% RSLogix 500 project SW2046_W.RSS, saved by version 11.00.00.00 %
PROJECT "PS7"    % processor: MicroLogix 1400 %

PROGRAM FILES
  LAD 2 "MAIN"  33 rungs  % Calls all system and subsystem routines %
  LAD 3 "CONSTANTS"  90 rungs  % Maintains the system constants %
  LAD 4 "DEFAULTS"  121 rungs  % Manages the system default values %
  LAD 5 "SYS_FAULTS"  58 rungs  % Monitors the system fault conditions %
  LAD 6 "SYSTEM"  93 rungs  % Controls the system %
  LAD 7 "PROCESSING"  14 rungs  % Runs the processing control %
  LAD 8 "MANUAL_CTL"  17 rungs  % Runs the manual valve control %
  LAD 9 "STARTUP"  25 rungs
  LAD 10 "PURIFY"  38 rungs  % Operates the purify control %
  LAD 11 "REGEN"  55 rungs  % Operates the regen control %
  LAD 12 "REGEN_FLT"  26 rungs  % regen alarms and warnings %
  LAD 13 "PURGE"  34 rungs
  LAD 14 "MFM"  5 rungs
  LAD 16 "MFC"  12 rungs
  LAD 17 "BYPASS"  4 rungs  % Controls the bypass %
  LAD 20 "ADS A"  46 rungs  % Controls the Adsorber A %
  LAD 21 "ADS A FLT"  18 rungs  % Controls the Adsorber A faults %
  LAD 22 "ADS B"  46 rungs  % Controld Adsorber B %
  LAD 23 "ADS B FLT"  17 rungs  % Controls the Adsorber B faults %
  LAD 24 "ADS PH"  10 rungs
  LAD 25 "ADS PH FLT"  15 rungs
  LAD 26 "GETTER"  24 rungs
  LAD 27 "GET 1 FLT"  15 rungs
  LAD 28 "GET 1"  25 rungs
  LAD 29 "GET 2 FLT"  15 rungs
  LAD 30 "GET 2"  25 rungs
  LAD 31 "GET 3 FLT"  15 rungs
  LAD 32 "GET 3"  25 rungs
  LAD 49 "MODBUS"  59 rungs
  LAD 50 "PLC FAULT"  7 rungs
  LAD 51 "REVERSE"  9 rungs
  LAD 252 "CLR_0034"  8 rungs

DATA FILES
  O0 OUTPUT  40 elements
  I1 INPUT  41 elements
  S2 STATUS  66 elements
  B3 BINARY  4 elements
  T4 TIMER  256 elements
  C5 COUNTER  256 elements
  R6 CONTROL  2 elements
  N7 SYSTEM CFG  120 elements  % Maintains the values that characterize the system %
  F8 FLOAT  8 elements
  N9 CONSTANTS  124 elements  % The collection of system and subsystem constants %
  N10 SYSTEM  36 elements  % Contain the values for system control %
  N11 PROCESS  4 elements  % Contains the values for the processing machine %
  N12 PURIFY  18 elements  % Contains the values required for purify %
  N13 REGEN  32 elements  % Contains the values required for regen %
  PD14 PID  10 elements
  N15 MANUAL CTL  5 elements  % Contains the data for the manual valve control %
  N16 ADSORBER_A  22 elements  % Contains the values for Adsorber A %
  N17 ADSORBER_B  22 elements  % Contains the values required for Adsorber B %
  N18 GETTER CMN  28 elements
  N19 BYPASS  2 elements
  N20 PURGE  10 elements
  N21 STARTUP  80 elements
  B22 STARTUP  6 elements
  N23 GETTER 1  15 elements
  N24 GETTER 2  15 elements
  N25 GETTER 3  15 elements
  B26 FAULTS  29 elements
  N27 NOMEMBCKUP  3 elements
  B29 GETTER  1 elements
  B30 SYSTEM CFG  6 elements
  B31 SYSTEM  10 elements
  B32 PROCESS  1 elements
  B33 PURIFY  1 elements
  B34 REGEN  3 elements
  B35 MANUAL CTL  3 elements
  B36 PURGE  2 elements
  L51 LONG  4 elements
  N55 TEST_START  5 elements  % Simultation Start %
  N64 MODBUS  126 elements
  MG68 COMMS  2 elements
  B69 REVERSE  3 elements
  N77 FAULT_FIFO  255 elements
  RIX81   1 elements
  N200   1 elements
  L201   1 elements
  L202   1 elements
  L203   2 elements
  F206   3 elements
  N207   6 elements
  N210   3 elements
  B250   1 elements
  T252   5 elements
  C253   6 elements

LADDER 2 "MAIN"    % Calls all system and subsystem routines %
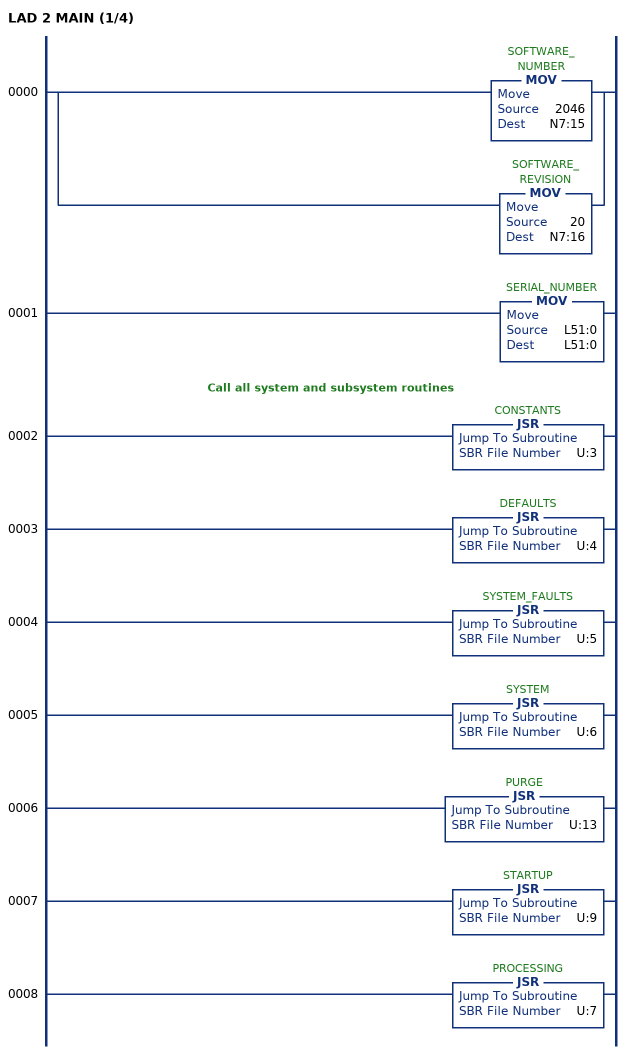
% Rung: 0 %
SOR BST MOV 2046 N7:15 NXB MOV 20 N7:16 BND EOR
%   N7:15  SOFTWARE_NUMBER %
%   N7:16  SOFTWARE_REVISION %
% Rung: 1 %
SOR MOV L51:0 L51:0 EOR
%   L51:0  SERIAL_NUMBER %
% Rung: 2 %
% TITLE: Call all system and subsystem routines %
SOR JSR U:3 EOR
%   U:3  CONSTANTS %
% Rung: 3 %
SOR JSR U:4 EOR
%   U:4  DEFAULTS %
% Rung: 4 %
SOR JSR U:5 EOR
%   U:5  SYSTEM_FAULTS %
% Rung: 5 %
SOR JSR U:6 EOR
%   U:6  SYSTEM %
% Rung: 6 %
SOR JSR U:13 EOR
%   U:13  PURGE %
% Rung: 7 %
SOR JSR U:9 EOR
%   U:9  STARTUP %
% Rung: 8 %
SOR JSR U:7 EOR
%   U:7  PROCESSING %

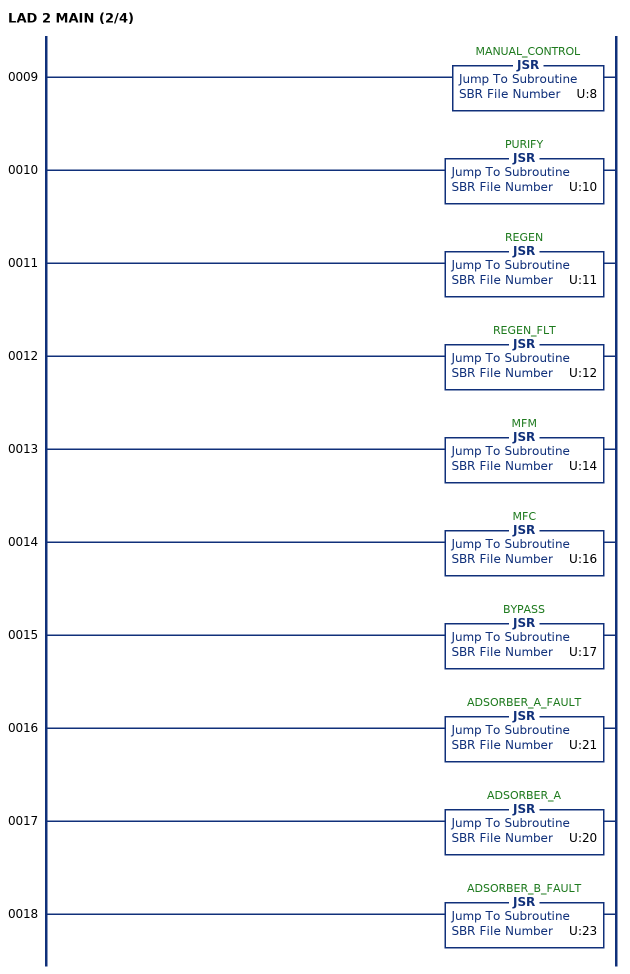
% Rung: 9 %
SOR JSR U:8 EOR
%   U:8  MANUAL_CONTROL %
% Rung: 10 %
SOR JSR U:10 EOR
%   U:10  PURIFY %
% Rung: 11 %
SOR JSR U:11 EOR
%   U:11  REGEN %
% Rung: 12 %
SOR JSR U:12 EOR
%   U:12  REGEN_FLT %
% Rung: 13 %
SOR JSR U:14 EOR
%   U:14  MFM %
% Rung: 14 %
SOR JSR U:16 EOR
%   U:16  MFC %
% Rung: 15 %
SOR JSR U:17 EOR
%   U:17  BYPASS %
% Rung: 16 %
SOR JSR U:21 EOR
%   U:21  ADSORBER_A_FAULT %
% Rung: 17 %
SOR JSR U:20 EOR
%   U:20  ADSORBER_A %
% Rung: 18 %
SOR JSR U:23 EOR
%   U:23  ADSORBER_B_FAULT %

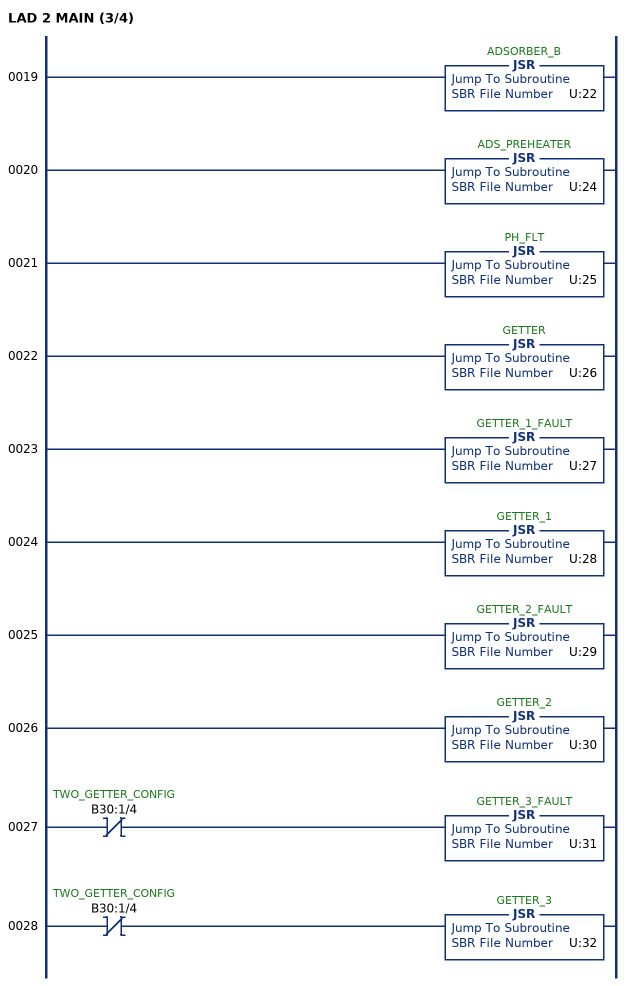
% Rung: 19 %
SOR JSR U:22 EOR
%   U:22  ADSORBER_B %
% Rung: 20 %
SOR JSR U:24 EOR
%   U:24  ADS_PREHEATER %
% Rung: 21 %
SOR JSR U:25 EOR
%   U:25  PH_FLT %
% Rung: 22 %
SOR JSR U:26 EOR
%   U:26  GETTER %
% Rung: 23 %
SOR JSR U:27 EOR
%   U:27  GETTER_1_FAULT %
% Rung: 24 %
SOR JSR U:28 EOR
%   U:28  GETTER_1 %
% Rung: 25 %
SOR JSR U:29 EOR
%   U:29  GETTER_2_FAULT %
% Rung: 26 %
SOR JSR U:30 EOR
%   U:30  GETTER_2 %
% Rung: 27 %
SOR XIO B30:1/4 JSR U:31 EOR
%   B30:1/4  TWO_GETTER_CONFIG %
%   U:31  GETTER_3_FAULT %
% Rung: 28 %
SOR XIO B30:1/4 JSR U:32 EOR
%   B30:1/4  TWO_GETTER_CONFIG %
%   U:32  GETTER_3 %

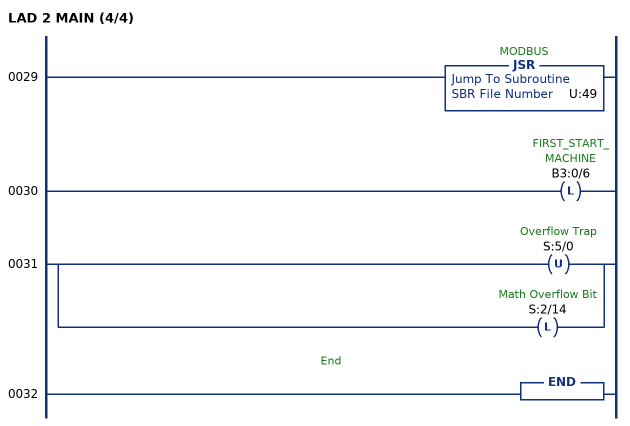
% Rung: 29 %
SOR JSR U:49 EOR
%   U:49  MODBUS %
% Rung: 30 %
SOR OTL B3:0/6 EOR
%   B3:0/6  FIRST_START_MACHINE %
% Rung: 31 %
SOR BST OTU S:5/0 NXB OTL S:2/14 BND EOR
%   S:5/0  "Overflow Trap" %
%   S:2/14  "Math Overflow Bit" %
% Rung: 32 %
% End %
SOR END EOR

LADDER 3 "CONSTANTS"    % Maintains the system constants %
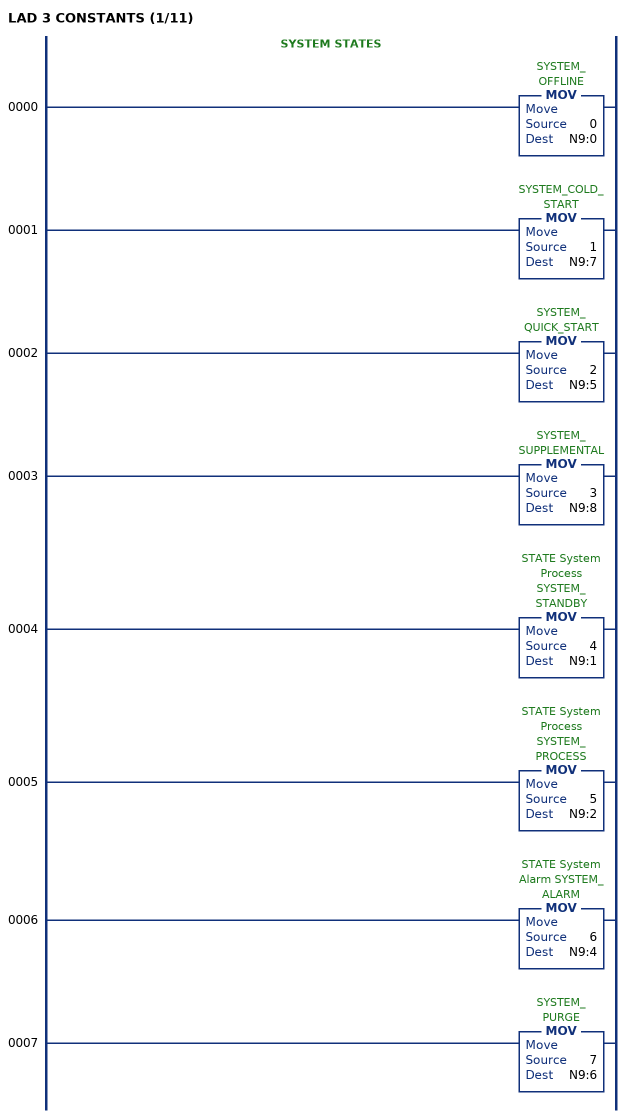
% Rung: 0 %
% TITLE: SYSTEM STATES %
SOR MOV 0 N9:0 EOR
%   N9:0  SYSTEM_OFFLINE %
% Rung: 1 %
SOR MOV 1 N9:7 EOR
%   N9:7  SYSTEM_COLD_START %
% Rung: 2 %
SOR MOV 2 N9:5 EOR
%   N9:5  SYSTEM_QUICK_START %
% Rung: 3 %
SOR MOV 3 N9:8 EOR
%   N9:8  SYSTEM_SUPPLEMENTAL %
% Rung: 4 %
SOR MOV 4 N9:1 EOR
%   N9:1  SYSTEM_STANDBY  "STATE System Process" %
% Rung: 5 %
SOR MOV 5 N9:2 EOR
%   N9:2  SYSTEM_PROCESS  "STATE System Process" %
% Rung: 6 %
SOR MOV 6 N9:4 EOR
%   N9:4  SYSTEM_ALARM  "STATE System Alarm" %
% Rung: 7 %
SOR MOV 7 N9:6 EOR
%   N9:6  SYSTEM_PURGE %

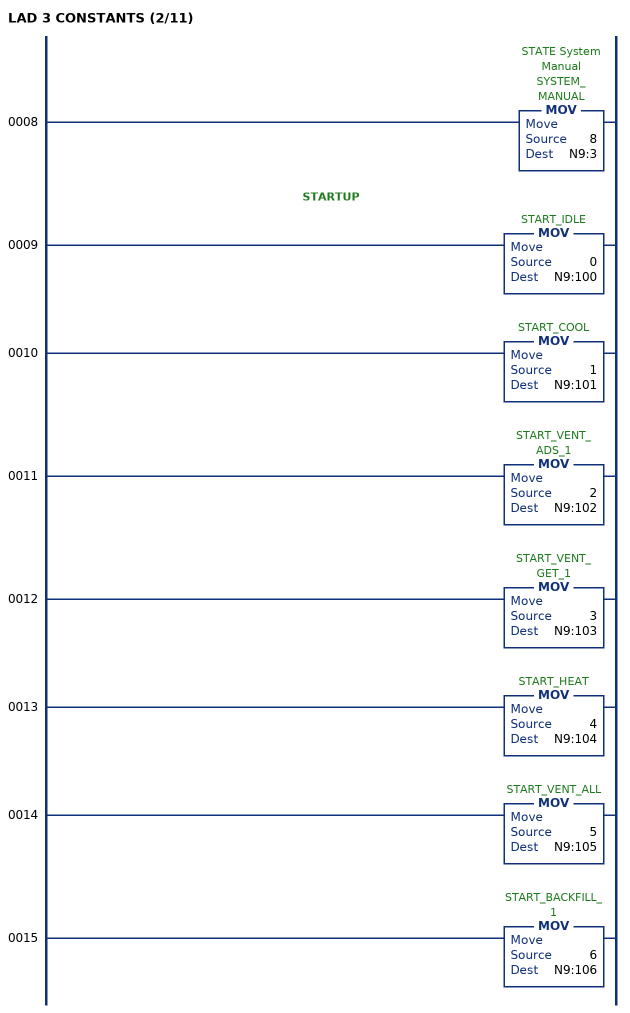
% Rung: 8 %
SOR MOV 8 N9:3 EOR
%   N9:3  SYSTEM_MANUAL  "STATE System Manual" %
% Rung: 9 %
% TITLE: STARTUP %
SOR MOV 0 N9:100 EOR
%   N9:100  START_IDLE %
% Rung: 10 %
SOR MOV 1 N9:101 EOR
%   N9:101  START_COOL %
% Rung: 11 %
SOR MOV 2 N9:102 EOR
%   N9:102  START_VENT_ADS_1 %
% Rung: 12 %
SOR MOV 3 N9:103 EOR
%   N9:103  START_VENT_GET_1 %
% Rung: 13 %
SOR MOV 4 N9:104 EOR
%   N9:104  START_HEAT %
% Rung: 14 %
SOR MOV 5 N9:105 EOR
%   N9:105  START_VENT_ALL %
% Rung: 15 %
SOR MOV 6 N9:106 EOR
%   N9:106  START_BACKFILL_1 %

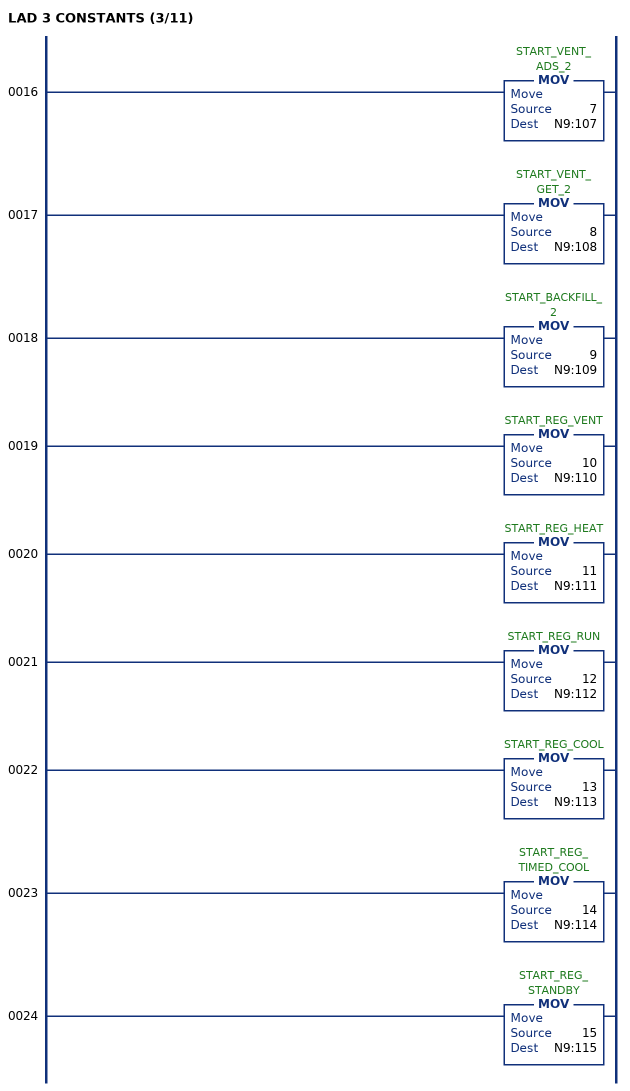
% Rung: 16 %
SOR MOV 7 N9:107 EOR
%   N9:107  START_VENT_ADS_2 %
% Rung: 17 %
SOR MOV 8 N9:108 EOR
%   N9:108  START_VENT_GET_2 %
% Rung: 18 %
SOR MOV 9 N9:109 EOR
%   N9:109  START_BACKFILL_2 %
% Rung: 19 %
SOR MOV 10 N9:110 EOR
%   N9:110  START_REG_VENT %
% Rung: 20 %
SOR MOV 11 N9:111 EOR
%   N9:111  START_REG_HEAT %
% Rung: 21 %
SOR MOV 12 N9:112 EOR
%   N9:112  START_REG_RUN %
% Rung: 22 %
SOR MOV 13 N9:113 EOR
%   N9:113  START_REG_COOL %
% Rung: 23 %
SOR MOV 14 N9:114 EOR
%   N9:114  START_REG_TIMED_COOL %
% Rung: 24 %
SOR MOV 15 N9:115 EOR
%   N9:115  START_REG_STANDBY %

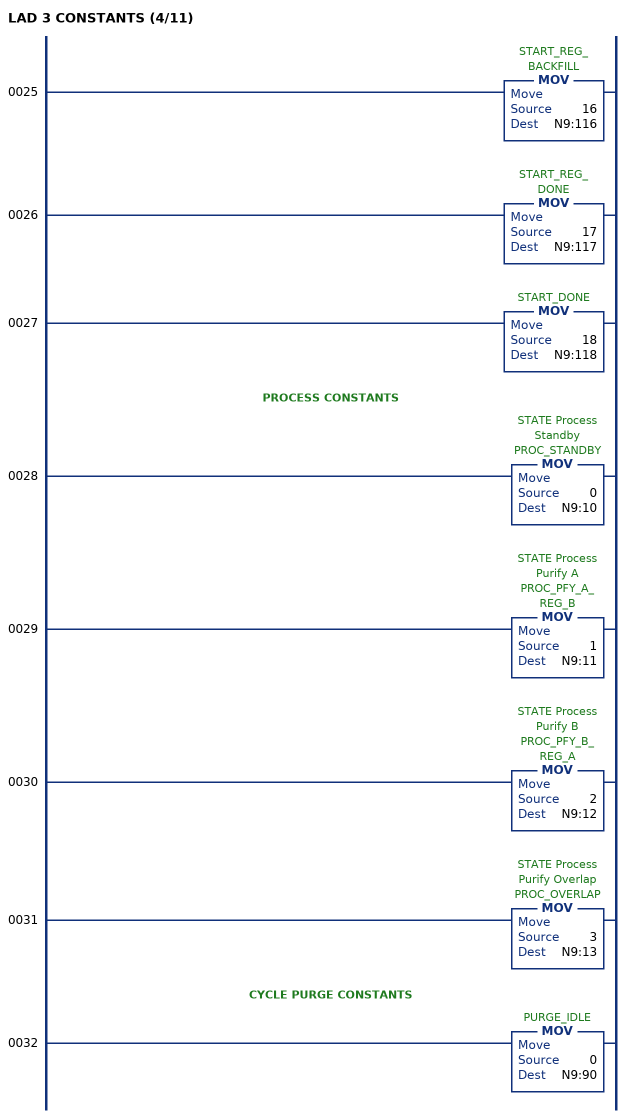
% Rung: 25 %
SOR MOV 16 N9:116 EOR
%   N9:116  START_REG_BACKFILL %
% Rung: 26 %
SOR MOV 17 N9:117 EOR
%   N9:117  START_REG_DONE %
% Rung: 27 %
SOR MOV 18 N9:118 EOR
%   N9:118  START_DONE %
% Rung: 28 %
% TITLE: PROCESS CONSTANTS %
SOR MOV 0 N9:10 EOR
%   N9:10  PROC_STANDBY  "STATE Process Standby" %
% Rung: 29 %
SOR MOV 1 N9:11 EOR
%   N9:11  PROC_PFY_A_REG_B  "STATE Process Purify A" %
% Rung: 30 %
SOR MOV 2 N9:12 EOR
%   N9:12  PROC_PFY_B_REG_A  "STATE Process Purify B" %
% Rung: 31 %
SOR MOV 3 N9:13 EOR
%   N9:13  PROC_OVERLAP  "STATE Process Purify Overlap" %
% Rung: 32 %
% TITLE: CYCLE PURGE CONSTANTS %
SOR MOV 0 N9:90 EOR
%   N9:90  PURGE_IDLE %

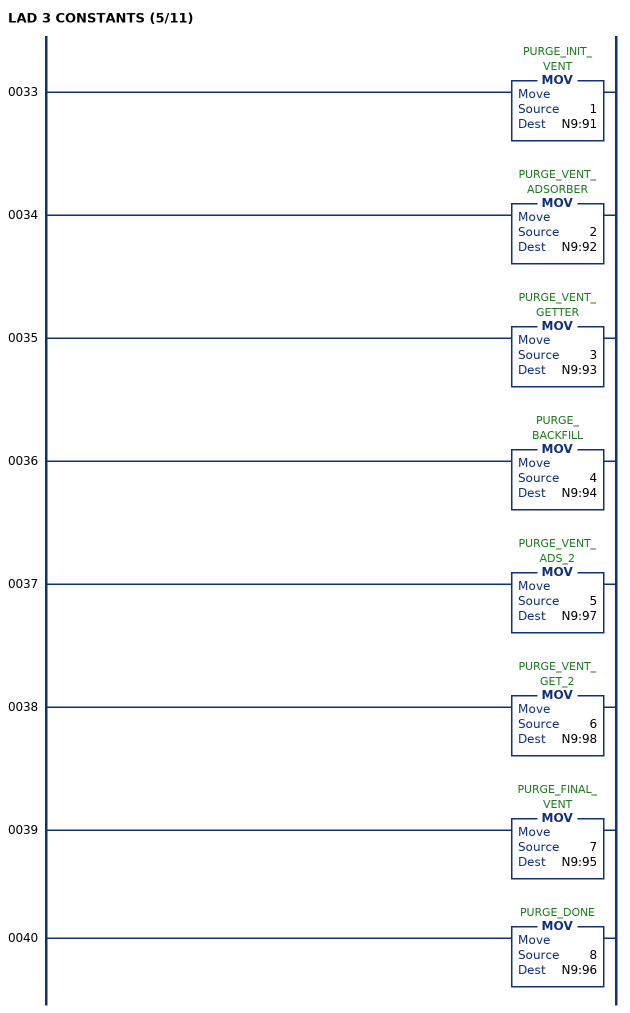
% Rung: 33 %
SOR MOV 1 N9:91 EOR
%   N9:91  PURGE_INIT_VENT %
% Rung: 34 %
SOR MOV 2 N9:92 EOR
%   N9:92  PURGE_VENT_ADSORBER %
% Rung: 35 %
SOR MOV 3 N9:93 EOR
%   N9:93  PURGE_VENT_GETTER %
% Rung: 36 %
SOR MOV 4 N9:94 EOR
%   N9:94  PURGE_BACKFILL %
% Rung: 37 %
SOR MOV 5 N9:97 EOR
%   N9:97  PURGE_VENT_ADS_2 %
% Rung: 38 %
SOR MOV 6 N9:98 EOR
%   N9:98  PURGE_VENT_GET_2 %
% Rung: 39 %
SOR MOV 7 N9:95 EOR
%   N9:95  PURGE_FINAL_VENT %
% Rung: 40 %
SOR MOV 8 N9:96 EOR
%   N9:96  PURGE_DONE %

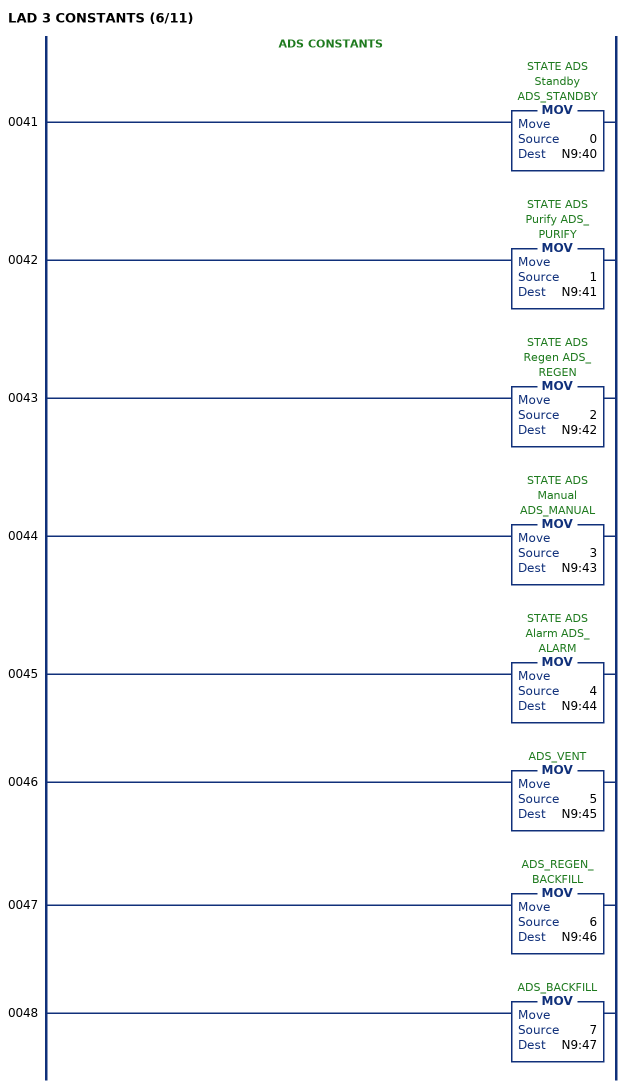
% Rung: 41 %
% TITLE: ADS CONSTANTS %
SOR MOV 0 N9:40 EOR
%   N9:40  ADS_STANDBY  "STATE ADS Standby" %
% Rung: 42 %
SOR MOV 1 N9:41 EOR
%   N9:41  ADS_PURIFY  "STATE ADS Purify" %
% Rung: 43 %
SOR MOV 2 N9:42 EOR
%   N9:42  ADS_REGEN  "STATE ADS Regen" %
% Rung: 44 %
SOR MOV 3 N9:43 EOR
%   N9:43  ADS_MANUAL  "STATE ADS Manual" %
% Rung: 45 %
SOR MOV 4 N9:44 EOR
%   N9:44  ADS_ALARM  "STATE ADS Alarm" %
% Rung: 46 %
SOR MOV 5 N9:45 EOR
%   N9:45  ADS_VENT %
% Rung: 47 %
SOR MOV 6 N9:46 EOR
%   N9:46  ADS_REGEN_BACKFILL %
% Rung: 48 %
SOR MOV 7 N9:47 EOR
%   N9:47  ADS_BACKFILL %

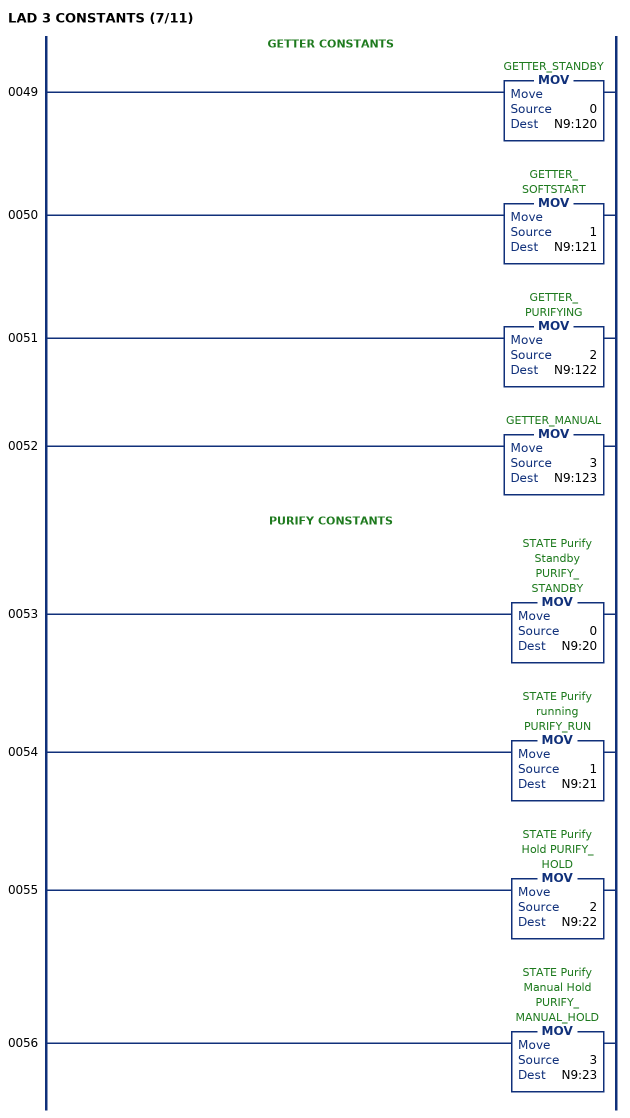
% Rung: 49 %
% TITLE: GETTER CONSTANTS %
SOR MOV 0 N9:120 EOR
%   N9:120  GETTER_STANDBY %
% Rung: 50 %
SOR MOV 1 N9:121 EOR
%   N9:121  GETTER_SOFTSTART %
% Rung: 51 %
SOR MOV 2 N9:122 EOR
%   N9:122  GETTER_PURIFYING %
% Rung: 52 %
SOR MOV 3 N9:123 EOR
%   N9:123  GETTER_MANUAL %
% Rung: 53 %
% TITLE: PURIFY CONSTANTS %
SOR MOV 0 N9:20 EOR
%   N9:20  PURIFY_STANDBY  "STATE Purify Standby" %
% Rung: 54 %
SOR MOV 1 N9:21 EOR
%   N9:21  PURIFY_RUN  "STATE Purify running" %
% Rung: 55 %
SOR MOV 2 N9:22 EOR
%   N9:22  PURIFY_HOLD  "STATE Purify Hold" %
% Rung: 56 %
SOR MOV 3 N9:23 EOR
%   N9:23  PURIFY_MANUAL_HOLD  "STATE Purify Manual Hold" %

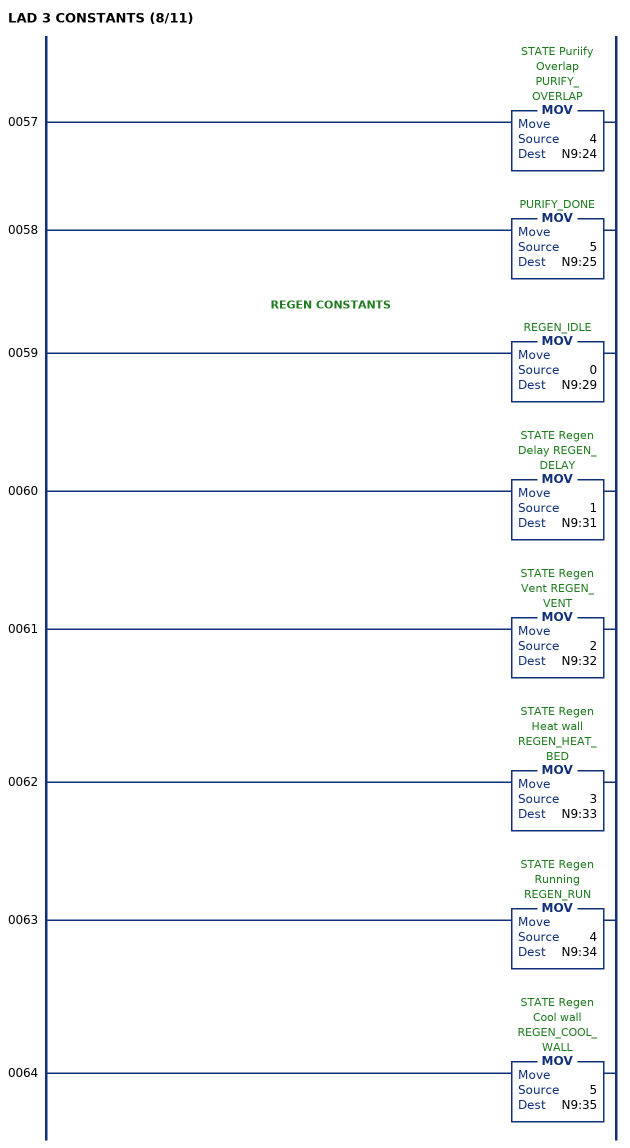
% Rung: 57 %
SOR MOV 4 N9:24 EOR
%   N9:24  PURIFY_OVERLAP  "STATE Puriify Overlap" %
% Rung: 58 %
SOR MOV 5 N9:25 EOR
%   N9:25  PURIFY_DONE %
% Rung: 59 %
% TITLE: REGEN CONSTANTS %
SOR MOV 0 N9:29 EOR
%   N9:29  REGEN_IDLE %
% Rung: 60 %
SOR MOV 1 N9:31 EOR
%   N9:31  REGEN_DELAY  "STATE Regen Delay" %
% Rung: 61 %
SOR MOV 2 N9:32 EOR
%   N9:32  REGEN_VENT  "STATE Regen Vent" %
% Rung: 62 %
SOR MOV 3 N9:33 EOR
%   N9:33  REGEN_HEAT_BED  "STATE Regen Heat wall" %
% Rung: 63 %
SOR MOV 4 N9:34 EOR
%   N9:34  REGEN_RUN  "STATE Regen Running" %
% Rung: 64 %
SOR MOV 5 N9:35 EOR
%   N9:35  REGEN_COOL_WALL  "STATE Regen Cool wall" %

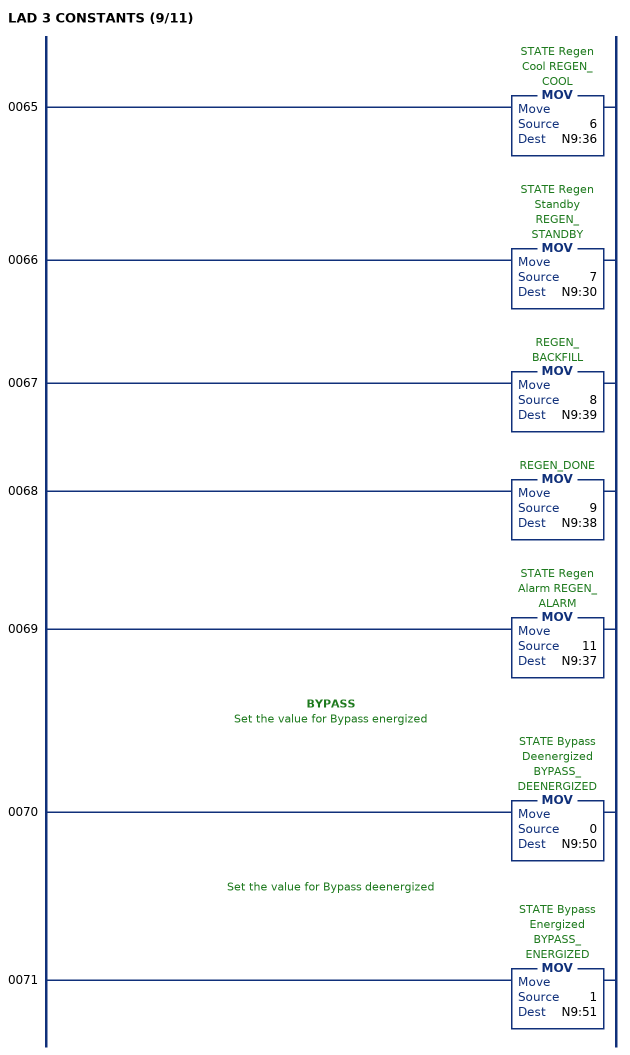
% Rung: 65 %
SOR MOV 6 N9:36 EOR
%   N9:36  REGEN_COOL  "STATE Regen Cool" %
% Rung: 66 %
SOR MOV 7 N9:30 EOR
%   N9:30  REGEN_STANDBY  "STATE Regen Standby" %
% Rung: 67 %
SOR MOV 8 N9:39 EOR
%   N9:39  REGEN_BACKFILL %
% Rung: 68 %
SOR MOV 9 N9:38 EOR
%   N9:38  REGEN_DONE %
% Rung: 69 %
SOR MOV 11 N9:37 EOR
%   N9:37  REGEN_ALARM  "STATE Regen Alarm" %
% Rung: 70 %
% TITLE: BYPASS %
% Set the value for Bypass energized %
SOR MOV 0 N9:50 EOR
%   N9:50  BYPASS_DEENERGIZED  "STATE Bypass Deenergized" %
% Rung: 71 %
% Set the value for Bypass deenergized %
SOR MOV 1 N9:51 EOR
%   N9:51  BYPASS_ENERGIZED  "STATE Bypass Energized" %

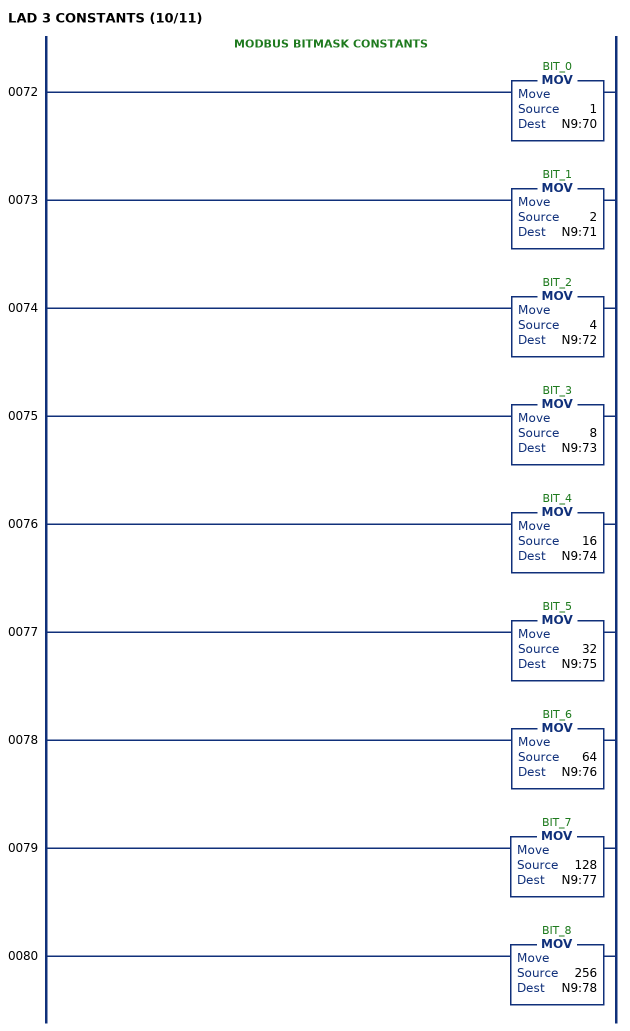
% Rung: 72 %
% TITLE: MODBUS BITMASK CONSTANTS %
SOR MOV 1 N9:70 EOR
%   N9:70  BIT_0 %
% Rung: 73 %
SOR MOV 2 N9:71 EOR
%   N9:71  BIT_1 %
% Rung: 74 %
SOR MOV 4 N9:72 EOR
%   N9:72  BIT_2 %
% Rung: 75 %
SOR MOV 8 N9:73 EOR
%   N9:73  BIT_3 %
% Rung: 76 %
SOR MOV 16 N9:74 EOR
%   N9:74  BIT_4 %
% Rung: 77 %
SOR MOV 32 N9:75 EOR
%   N9:75  BIT_5 %
% Rung: 78 %
SOR MOV 64 N9:76 EOR
%   N9:76  BIT_6 %
% Rung: 79 %
SOR MOV 128 N9:77 EOR
%   N9:77  BIT_7 %
% Rung: 80 %
SOR MOV 256 N9:78 EOR
%   N9:78  BIT_8 %

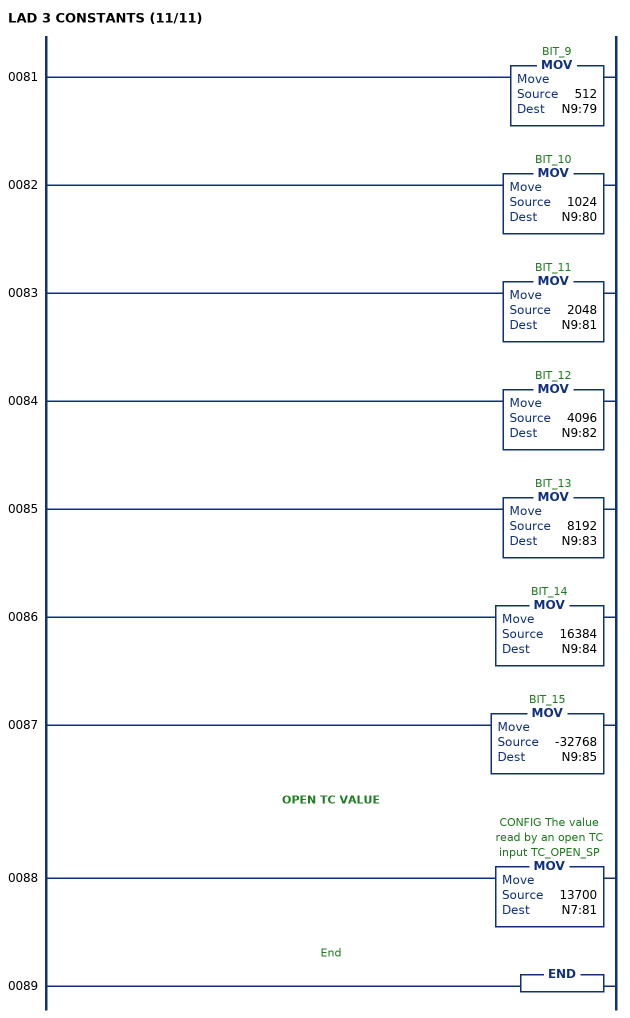
% Rung: 81 %
SOR MOV 512 N9:79 EOR
%   N9:79  BIT_9 %
% Rung: 82 %
SOR MOV 1024 N9:80 EOR
%   N9:80  BIT_10 %
% Rung: 83 %
SOR MOV 2048 N9:81 EOR
%   N9:81  BIT_11 %
% Rung: 84 %
SOR MOV 4096 N9:82 EOR
%   N9:82  BIT_12 %
% Rung: 85 %
SOR MOV 8192 N9:83 EOR
%   N9:83  BIT_13 %
% Rung: 86 %
SOR MOV 16384 N9:84 EOR
%   N9:84  BIT_14 %
% Rung: 87 %
SOR MOV -32768 N9:85 EOR
%   N9:85  BIT_15 %
% Rung: 88 %
% TITLE: OPEN TC VALUE %
SOR MOV 13700 N7:81 EOR
%   N7:81  TC_OPEN_SP  "CONFIG The value read by an open TC input" %
% Rung: 89 %
% End %
SOR END EOR

LADDER 4 "DEFAULTS"    % Manages the system default values %
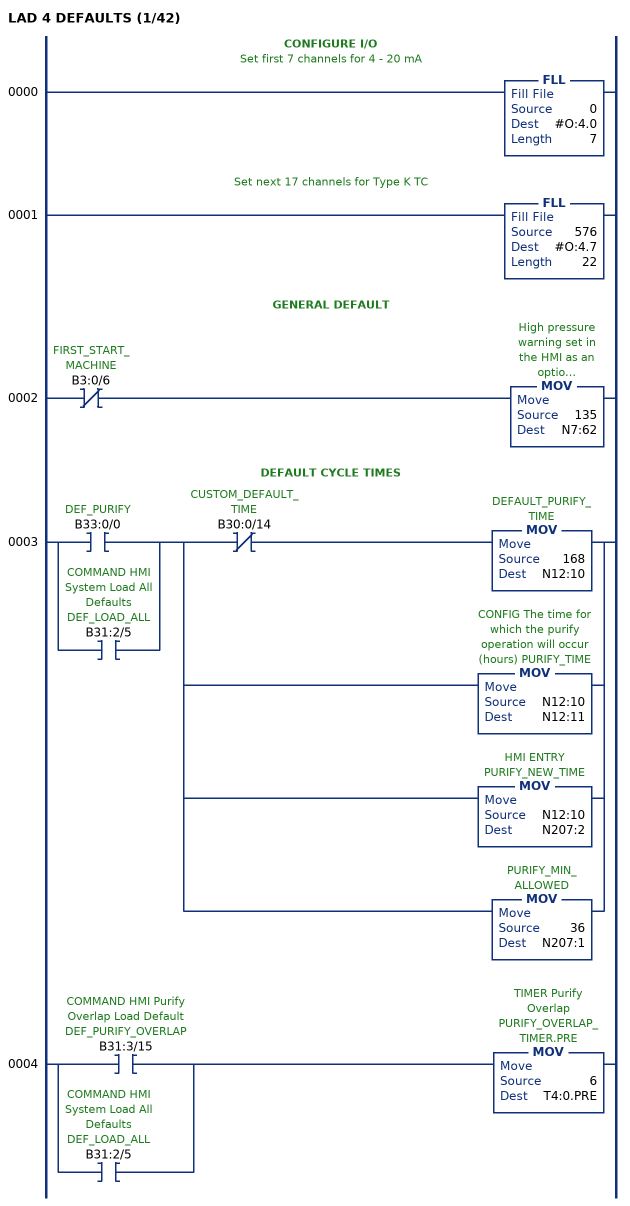
% Rung: 0 %
% TITLE: CONFIGURE I/O %
% Set first 7 channels for 4 - 20 mA %
SOR FLL 0 #O:4.0 7 EOR
% Rung: 1 %
% Set next 17 channels for Type K TC %
SOR FLL 576 #O:4.7 22 EOR
% Rung: 2 %
% TITLE: GENERAL DEFAULT %
SOR XIO B3:0/6 MOV 135 N7:62 EOR
%   B3:0/6  FIRST_START_MACHINE %
%   N7:62  HP_GAS_WRN_HMI_SP  "High pressure warning set in the HMI as an option" %
% Rung: 3 %
% TITLE: DEFAULT CYCLE TIMES %
SOR BST XIC B33:0/0 NXB XIC B31:2/5 BND BST XIO B30:0/14 MOV 168 N12:10 NXB MOV N12:10 N12:11 NXB MOV N12:10 N207:2 NXB MOV 36 N207:1 BND EOR
%   B33:0/0  DEF_PURIFY %
%   B31:2/5  DEF_LOAD_ALL  "COMMAND HMI System Load All Defaults" %
%   B30:0/14  CUSTOM_DEFAULT_TIME %
%   N12:10  DEFAULT_PURIFY_TIME %
%   N12:11  PURIFY_TIME  "CONFIG The time for which the purify operation will occur (hours)" %
%   N207:2  PURIFY_NEW_TIME  "HMI ENTRY" %
%   N207:1  PURIFY_MIN_ALLOWED %
% Rung: 4 %
SOR BST XIC B31:3/15 NXB XIC B31:2/5 BND MOV 6 T4:0.PRE EOR
%   B31:3/15  DEF_PURIFY_OVERLAP  "COMMAND HMI Purify Overlap Load Default" %
%   B31:2/5  DEF_LOAD_ALL  "COMMAND HMI System Load All Defaults" %
%   T4:0  PURIFY_OVERLAP_TIMER  "TIMER Purify Overlap" %

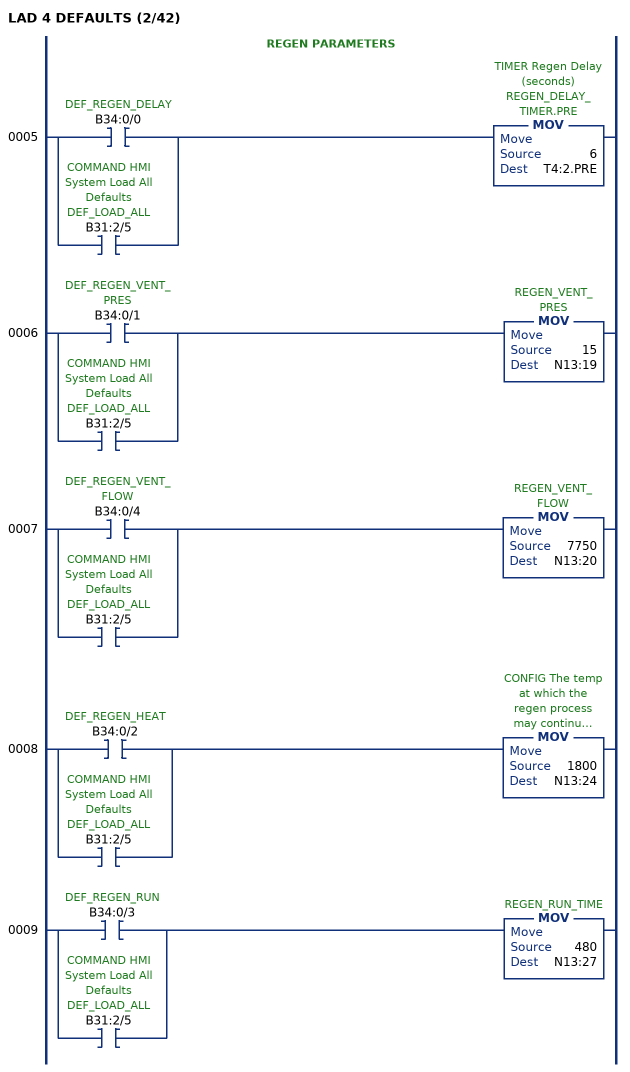
% Rung: 5 %
% TITLE: REGEN PARAMETERS %
SOR BST XIC B34:0/0 NXB XIC B31:2/5 BND MOV 6 T4:2.PRE EOR
%   B34:0/0  DEF_REGEN_DELAY %
%   B31:2/5  DEF_LOAD_ALL  "COMMAND HMI System Load All Defaults" %
%   T4:2  REGEN_DELAY_TIMER  "TIMER Regen Delay (seconds)" %
% Rung: 6 %
SOR BST XIC B34:0/1 NXB XIC B31:2/5 BND MOV 15 N13:19 EOR
%   B34:0/1  DEF_REGEN_VENT_PRES %
%   B31:2/5  DEF_LOAD_ALL  "COMMAND HMI System Load All Defaults" %
%   N13:19  REGEN_VENT_PRES %
% Rung: 7 %
SOR BST XIC B34:0/4 NXB XIC B31:2/5 BND MOV 7750 N13:20 EOR
%   B34:0/4  DEF_REGEN_VENT_FLOW %
%   B31:2/5  DEF_LOAD_ALL  "COMMAND HMI System Load All Defaults" %
%   N13:20  REGEN_VENT_FLOW %
% Rung: 8 %
SOR BST XIC B34:0/2 NXB XIC B31:2/5 BND MOV 1800 N13:24 EOR
%   B34:0/2  DEF_REGEN_HEAT %
%   B31:2/5  DEF_LOAD_ALL  "COMMAND HMI System Load All Defaults" %
%   N13:24  ADS_BED_TEMP_HIGH  "CONFIG The temp at which the regen process may continue" %
% Rung: 9 %
SOR BST XIC B34:0/3 NXB XIC B31:2/5 BND MOV 480 N13:27 EOR
%   B34:0/3  DEF_REGEN_RUN %
%   B31:2/5  DEF_LOAD_ALL  "COMMAND HMI System Load All Defaults" %
%   N13:27  REGEN_RUN_TIME %

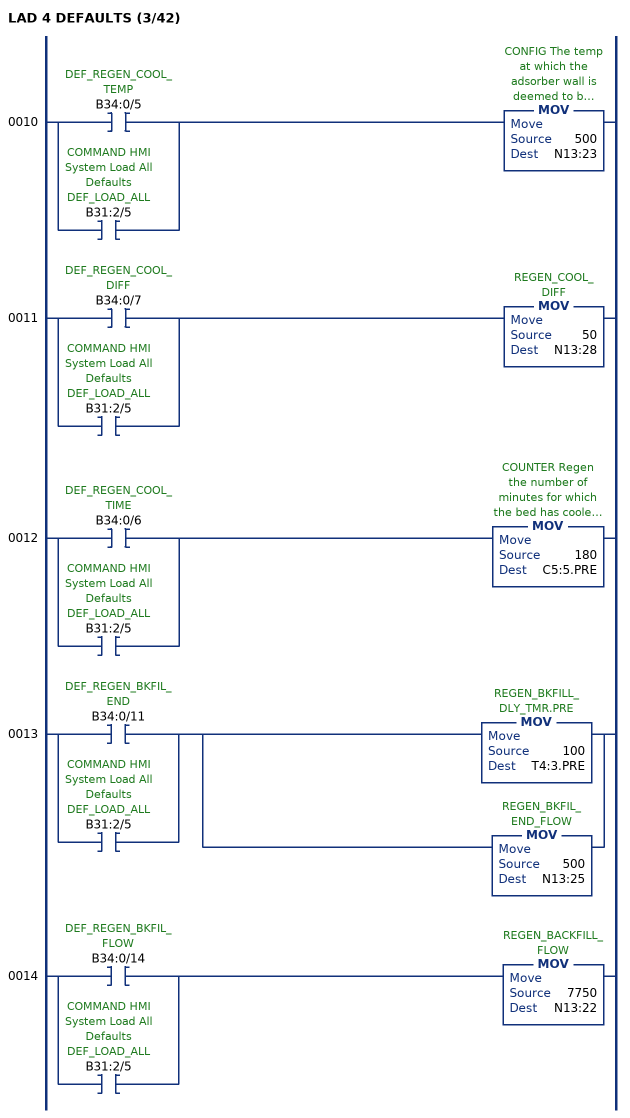
% Rung: 10 %
SOR BST XIC B34:0/5 NXB XIC B31:2/5 BND MOV 500 N13:23 EOR
%   B34:0/5  DEF_REGEN_COOL_TEMP %
%   B31:2/5  DEF_LOAD_ALL  "COMMAND HMI System Load All Defaults" %
%   N13:23  ADS_WALL_TEMP_COOL  "CONFIG The temp at which the adsorber wall is deemed to be cool enough to purify" %
% Rung: 11 %
SOR BST XIC B34:0/7 NXB XIC B31:2/5 BND MOV 50 N13:28 EOR
%   B34:0/7  DEF_REGEN_COOL_DIFF %
%   B31:2/5  DEF_LOAD_ALL  "COMMAND HMI System Load All Defaults" %
%   N13:28  REGEN_COOL_DIFF %
% Rung: 12 %
SOR BST XIC B34:0/6 NXB XIC B31:2/5 BND MOV 180 C5:5.PRE EOR
%   B34:0/6  DEF_REGEN_COOL_TIME %
%   B31:2/5  DEF_LOAD_ALL  "COMMAND HMI System Load All Defaults" %
%   C5:5  REGEN_COOL_MINUTE  "COUNTER Regen the number of minutes for which the bed has cooled" %
% Rung: 13 %
SOR BST XIC B34:0/11 NXB XIC B31:2/5 BND BST MOV 100 T4:3.PRE NXB MOV 500 N13:25 BND EOR
%   B34:0/11  DEF_REGEN_BKFIL_END %
%   B31:2/5  DEF_LOAD_ALL  "COMMAND HMI System Load All Defaults" %
%   T4:3  REGEN_BKFILL_DLY_TMR %
%   N13:25  REGEN_BKFIL_END_FLOW %
% Rung: 14 %
SOR BST XIC B34:0/14 NXB XIC B31:2/5 BND MOV 7750 N13:22 EOR
%   B34:0/14  DEF_REGEN_BKFIL_FLOW %
%   B31:2/5  DEF_LOAD_ALL  "COMMAND HMI System Load All Defaults" %
%   N13:22  REGEN_BACKFILL_FLOW %

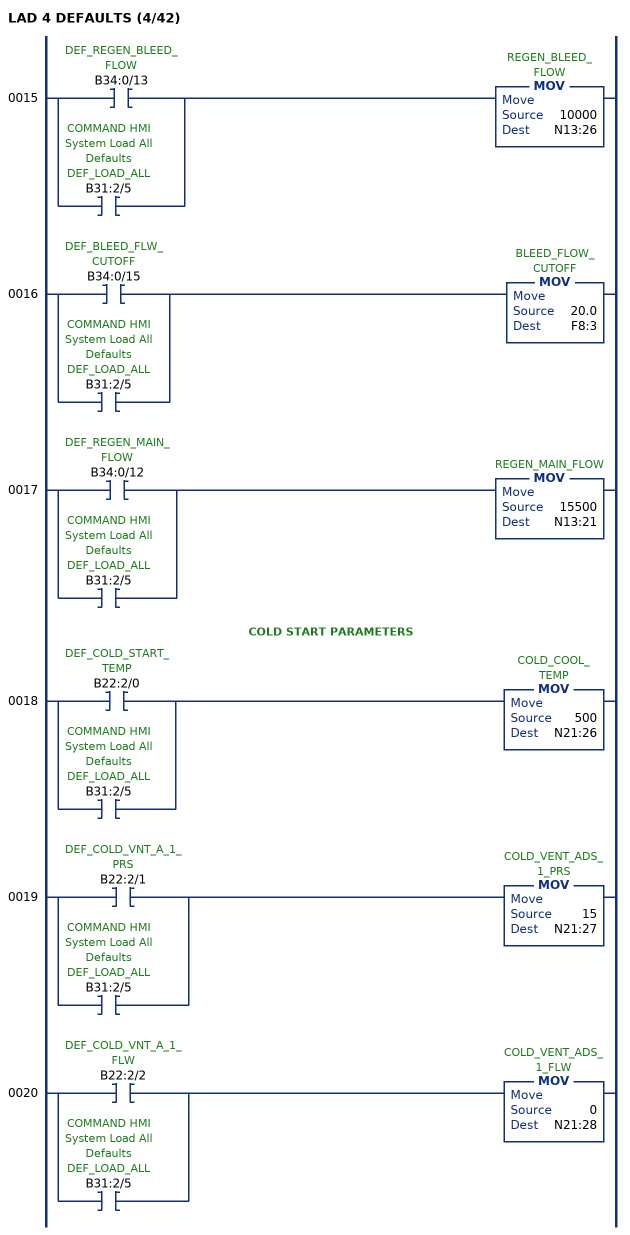
% Rung: 15 %
SOR BST XIC B34:0/13 NXB XIC B31:2/5 BND MOV 10000 N13:26 EOR
%   B34:0/13  DEF_REGEN_BLEED_FLOW %
%   B31:2/5  DEF_LOAD_ALL  "COMMAND HMI System Load All Defaults" %
%   N13:26  REGEN_BLEED_FLOW %
% Rung: 16 %
SOR BST XIC B34:0/15 NXB XIC B31:2/5 BND MOV 20.0 F8:3 EOR
%   B34:0/15  DEF_BLEED_FLW_CUTOFF %
%   B31:2/5  DEF_LOAD_ALL  "COMMAND HMI System Load All Defaults" %
%   F8:3  BLEED_FLOW_CUTOFF %
% Rung: 17 %
SOR BST XIC B34:0/12 NXB XIC B31:2/5 BND MOV 15500 N13:21 EOR
%   B34:0/12  DEF_REGEN_MAIN_FLOW %
%   B31:2/5  DEF_LOAD_ALL  "COMMAND HMI System Load All Defaults" %
%   N13:21  REGEN_MAIN_FLOW %
% Rung: 18 %
% TITLE: COLD START PARAMETERS %
SOR BST XIC B22:2/0 NXB XIC B31:2/5 BND MOV 500 N21:26 EOR
%   B22:2/0  DEF_COLD_START_TEMP %
%   B31:2/5  DEF_LOAD_ALL  "COMMAND HMI System Load All Defaults" %
%   N21:26  COLD_COOL_TEMP %
% Rung: 19 %
SOR BST XIC B22:2/1 NXB XIC B31:2/5 BND MOV 15 N21:27 EOR
%   B22:2/1  DEF_COLD_VNT_A_1_PRS %
%   B31:2/5  DEF_LOAD_ALL  "COMMAND HMI System Load All Defaults" %
%   N21:27  COLD_VENT_ADS_1_PRS %
% Rung: 20 %
SOR BST XIC B22:2/2 NXB XIC B31:2/5 BND MOV 0 N21:28 EOR
%   B22:2/2  DEF_COLD_VNT_A_1_FLW %
%   B31:2/5  DEF_LOAD_ALL  "COMMAND HMI System Load All Defaults" %
%   N21:28  COLD_VENT_ADS_1_FLW %

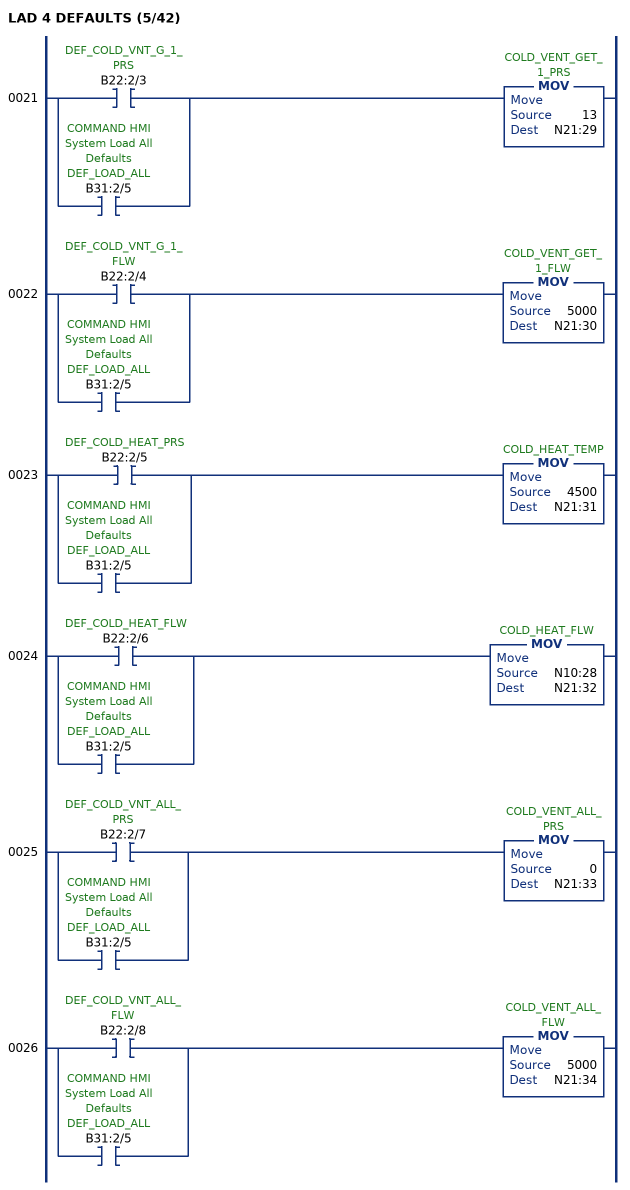
% Rung: 21 %
SOR BST XIC B22:2/3 NXB XIC B31:2/5 BND MOV 13 N21:29 EOR
%   B22:2/3  DEF_COLD_VNT_G_1_PRS %
%   B31:2/5  DEF_LOAD_ALL  "COMMAND HMI System Load All Defaults" %
%   N21:29  COLD_VENT_GET_1_PRS %
% Rung: 22 %
SOR BST XIC B22:2/4 NXB XIC B31:2/5 BND MOV 5000 N21:30 EOR
%   B22:2/4  DEF_COLD_VNT_G_1_FLW %
%   B31:2/5  DEF_LOAD_ALL  "COMMAND HMI System Load All Defaults" %
%   N21:30  COLD_VENT_GET_1_FLW %
% Rung: 23 %
SOR BST XIC B22:2/5 NXB XIC B31:2/5 BND MOV 4500 N21:31 EOR
%   B22:2/5  DEF_COLD_HEAT_PRS %
%   B31:2/5  DEF_LOAD_ALL  "COMMAND HMI System Load All Defaults" %
%   N21:31  COLD_HEAT_TEMP %
% Rung: 24 %
SOR BST XIC B22:2/6 NXB XIC B31:2/5 BND MOV N10:28 N21:32 EOR
%   B22:2/6  DEF_COLD_HEAT_FLW %
%   B31:2/5  DEF_LOAD_ALL  "COMMAND HMI System Load All Defaults" %
%   N10:28  MFC_SCALING  "in slpm" %
%   N21:32  COLD_HEAT_FLW %
% Rung: 25 %
SOR BST XIC B22:2/7 NXB XIC B31:2/5 BND MOV 0 N21:33 EOR
%   B22:2/7  DEF_COLD_VNT_ALL_PRS %
%   B31:2/5  DEF_LOAD_ALL  "COMMAND HMI System Load All Defaults" %
%   N21:33  COLD_VENT_ALL_PRS %
% Rung: 26 %
SOR BST XIC B22:2/8 NXB XIC B31:2/5 BND MOV 5000 N21:34 EOR
%   B22:2/8  DEF_COLD_VNT_ALL_FLW %
%   B31:2/5  DEF_LOAD_ALL  "COMMAND HMI System Load All Defaults" %
%   N21:34  COLD_VENT_ALL_FLW %

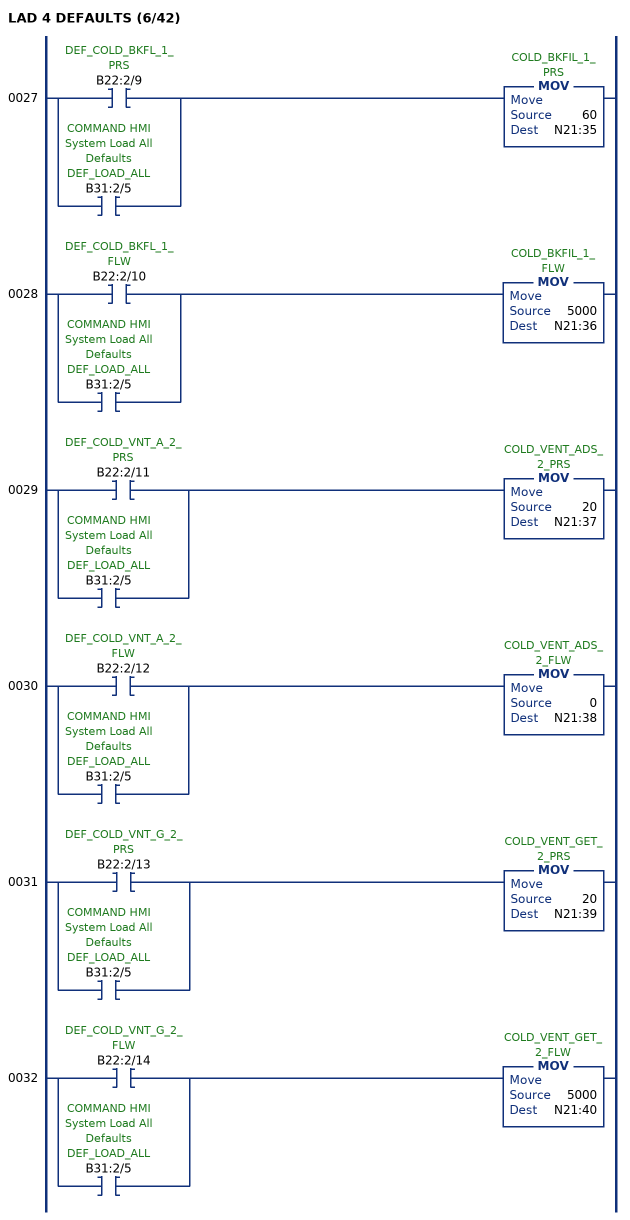
% Rung: 27 %
SOR BST XIC B22:2/9 NXB XIC B31:2/5 BND MOV 60 N21:35 EOR
%   B22:2/9  DEF_COLD_BKFL_1_PRS %
%   B31:2/5  DEF_LOAD_ALL  "COMMAND HMI System Load All Defaults" %
%   N21:35  COLD_BKFIL_1_PRS %
% Rung: 28 %
SOR BST XIC B22:2/10 NXB XIC B31:2/5 BND MOV 5000 N21:36 EOR
%   B22:2/10  DEF_COLD_BKFL_1_FLW %
%   B31:2/5  DEF_LOAD_ALL  "COMMAND HMI System Load All Defaults" %
%   N21:36  COLD_BKFIL_1_FLW %
% Rung: 29 %
SOR BST XIC B22:2/11 NXB XIC B31:2/5 BND MOV 20 N21:37 EOR
%   B22:2/11  DEF_COLD_VNT_A_2_PRS %
%   B31:2/5  DEF_LOAD_ALL  "COMMAND HMI System Load All Defaults" %
%   N21:37  COLD_VENT_ADS_2_PRS %
% Rung: 30 %
SOR BST XIC B22:2/12 NXB XIC B31:2/5 BND MOV 0 N21:38 EOR
%   B22:2/12  DEF_COLD_VNT_A_2_FLW %
%   B31:2/5  DEF_LOAD_ALL  "COMMAND HMI System Load All Defaults" %
%   N21:38  COLD_VENT_ADS_2_FLW %
% Rung: 31 %
SOR BST XIC B22:2/13 NXB XIC B31:2/5 BND MOV 20 N21:39 EOR
%   B22:2/13  DEF_COLD_VNT_G_2_PRS %
%   B31:2/5  DEF_LOAD_ALL  "COMMAND HMI System Load All Defaults" %
%   N21:39  COLD_VENT_GET_2_PRS %
% Rung: 32 %
SOR BST XIC B22:2/14 NXB XIC B31:2/5 BND MOV 5000 N21:40 EOR
%   B22:2/14  DEF_COLD_VNT_G_2_FLW %
%   B31:2/5  DEF_LOAD_ALL  "COMMAND HMI System Load All Defaults" %
%   N21:40  COLD_VENT_GET_2_FLW %

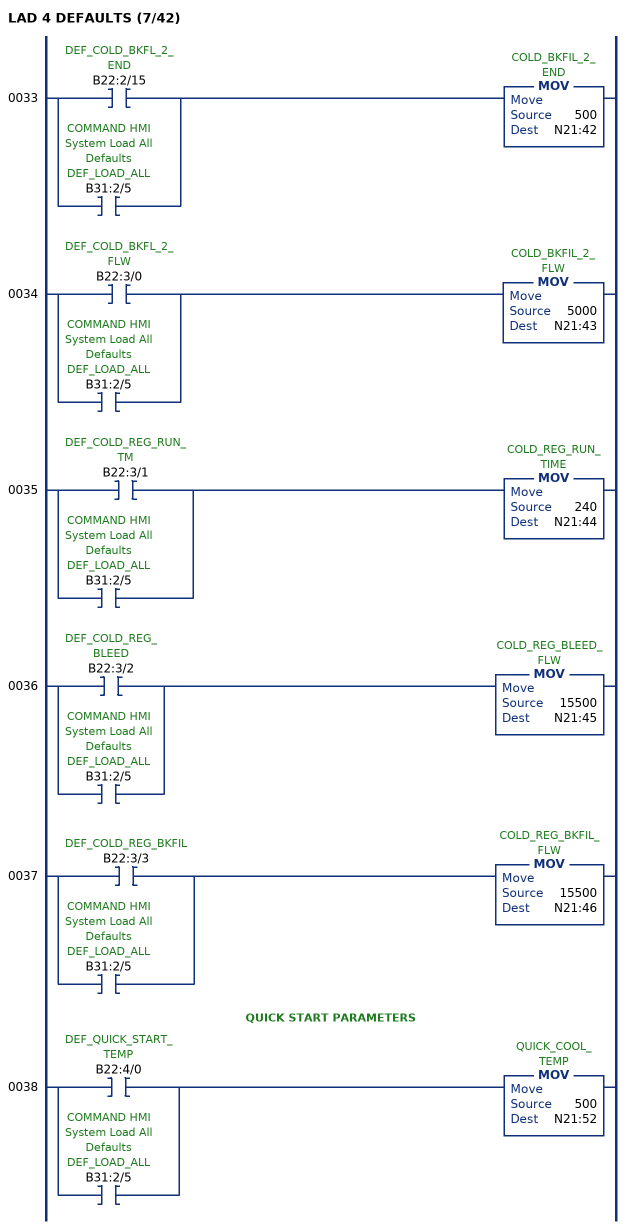
% Rung: 33 %
SOR BST XIC B22:2/15 NXB XIC B31:2/5 BND MOV 500 N21:42 EOR
%   B22:2/15  DEF_COLD_BKFL_2_END %
%   B31:2/5  DEF_LOAD_ALL  "COMMAND HMI System Load All Defaults" %
%   N21:42  COLD_BKFIL_2_END %
% Rung: 34 %
SOR BST XIC B22:3/0 NXB XIC B31:2/5 BND MOV 5000 N21:43 EOR
%   B22:3/0  DEF_COLD_BKFL_2_FLW %
%   B31:2/5  DEF_LOAD_ALL  "COMMAND HMI System Load All Defaults" %
%   N21:43  COLD_BKFIL_2_FLW %
% Rung: 35 %
SOR BST XIC B22:3/1 NXB XIC B31:2/5 BND MOV 240 N21:44 EOR
%   B22:3/1  DEF_COLD_REG_RUN_TM %
%   B31:2/5  DEF_LOAD_ALL  "COMMAND HMI System Load All Defaults" %
%   N21:44  COLD_REG_RUN_TIME %
% Rung: 36 %
SOR BST XIC B22:3/2 NXB XIC B31:2/5 BND MOV 15500 N21:45 EOR
%   B22:3/2  DEF_COLD_REG_BLEED %
%   B31:2/5  DEF_LOAD_ALL  "COMMAND HMI System Load All Defaults" %
%   N21:45  COLD_REG_BLEED_FLW %
% Rung: 37 %
SOR BST XIC B22:3/3 NXB XIC B31:2/5 BND MOV 15500 N21:46 EOR
%   B22:3/3  DEF_COLD_REG_BKFIL %
%   B31:2/5  DEF_LOAD_ALL  "COMMAND HMI System Load All Defaults" %
%   N21:46  COLD_REG_BKFIL_FLW %
% Rung: 38 %
% TITLE: QUICK START PARAMETERS %
SOR BST XIC B22:4/0 NXB XIC B31:2/5 BND MOV 500 N21:52 EOR
%   B22:4/0  DEF_QUICK_START_TEMP %
%   B31:2/5  DEF_LOAD_ALL  "COMMAND HMI System Load All Defaults" %
%   N21:52  QUICK_COOL_TEMP %

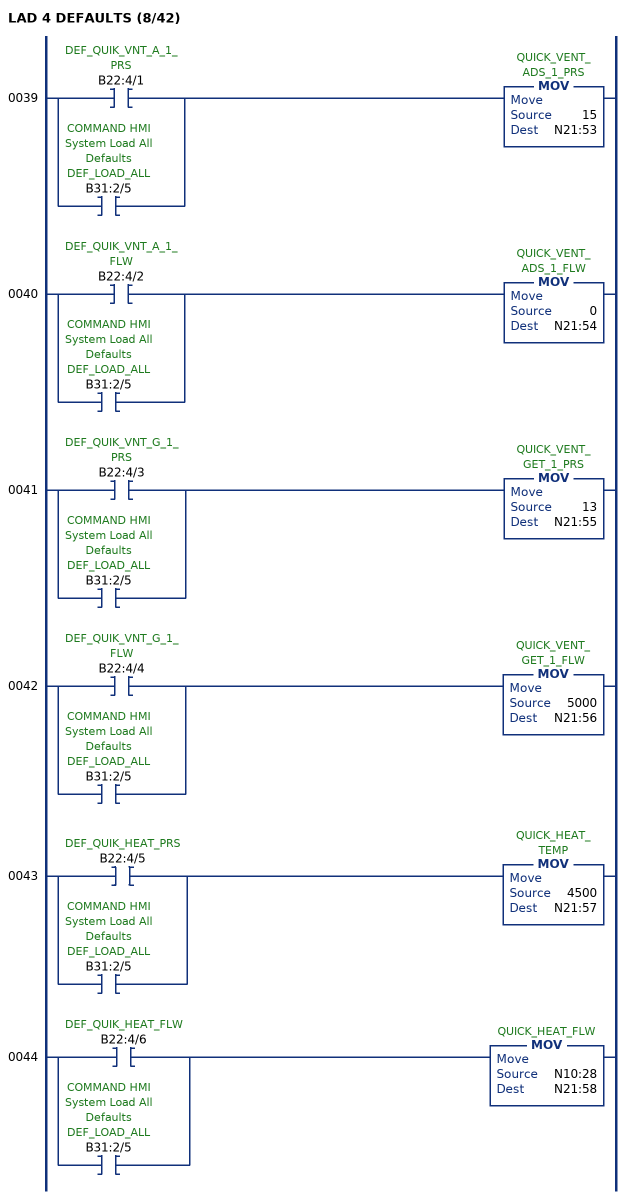
% Rung: 39 %
SOR BST XIC B22:4/1 NXB XIC B31:2/5 BND MOV 15 N21:53 EOR
%   B22:4/1  DEF_QUIK_VNT_A_1_PRS %
%   B31:2/5  DEF_LOAD_ALL  "COMMAND HMI System Load All Defaults" %
%   N21:53  QUICK_VENT_ADS_1_PRS %
% Rung: 40 %
SOR BST XIC B22:4/2 NXB XIC B31:2/5 BND MOV 0 N21:54 EOR
%   B22:4/2  DEF_QUIK_VNT_A_1_FLW %
%   B31:2/5  DEF_LOAD_ALL  "COMMAND HMI System Load All Defaults" %
%   N21:54  QUICK_VENT_ADS_1_FLW %
% Rung: 41 %
SOR BST XIC B22:4/3 NXB XIC B31:2/5 BND MOV 13 N21:55 EOR
%   B22:4/3  DEF_QUIK_VNT_G_1_PRS %
%   B31:2/5  DEF_LOAD_ALL  "COMMAND HMI System Load All Defaults" %
%   N21:55  QUICK_VENT_GET_1_PRS %
% Rung: 42 %
SOR BST XIC B22:4/4 NXB XIC B31:2/5 BND MOV 5000 N21:56 EOR
%   B22:4/4  DEF_QUIK_VNT_G_1_FLW %
%   B31:2/5  DEF_LOAD_ALL  "COMMAND HMI System Load All Defaults" %
%   N21:56  QUICK_VENT_GET_1_FLW %
% Rung: 43 %
SOR BST XIC B22:4/5 NXB XIC B31:2/5 BND MOV 4500 N21:57 EOR
%   B22:4/5  DEF_QUIK_HEAT_PRS %
%   B31:2/5  DEF_LOAD_ALL  "COMMAND HMI System Load All Defaults" %
%   N21:57  QUICK_HEAT_TEMP %
% Rung: 44 %
SOR BST XIC B22:4/6 NXB XIC B31:2/5 BND MOV N10:28 N21:58 EOR
%   B22:4/6  DEF_QUIK_HEAT_FLW %
%   B31:2/5  DEF_LOAD_ALL  "COMMAND HMI System Load All Defaults" %
%   N10:28  MFC_SCALING  "in slpm" %
%   N21:58  QUICK_HEAT_FLW %

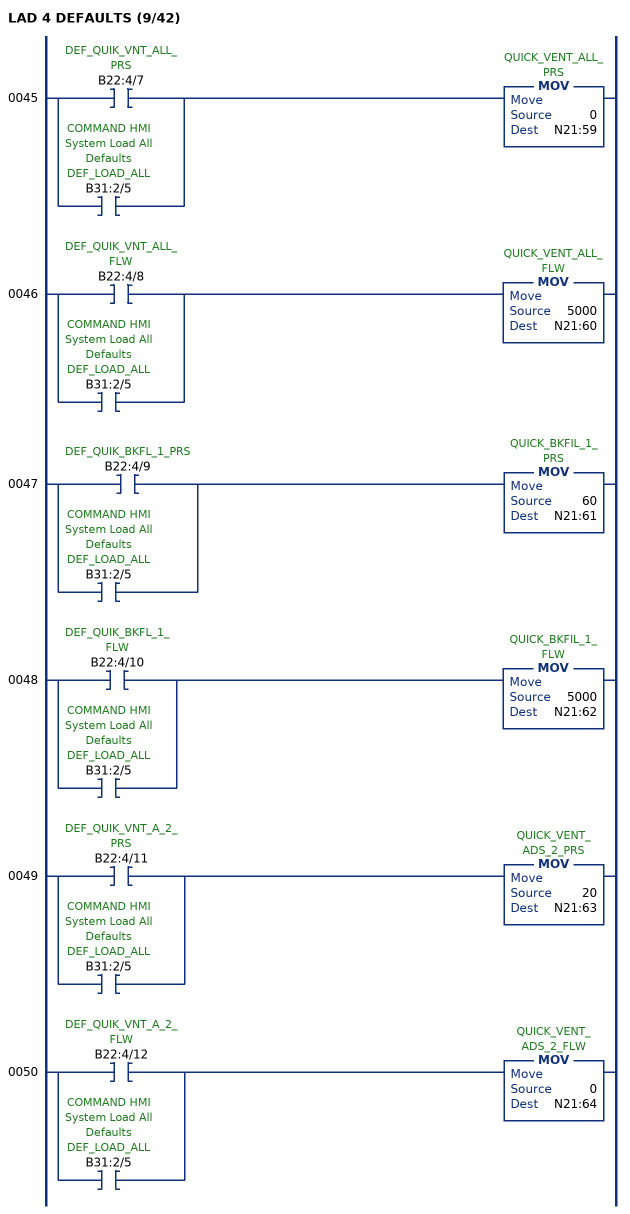
% Rung: 45 %
SOR BST XIC B22:4/7 NXB XIC B31:2/5 BND MOV 0 N21:59 EOR
%   B22:4/7  DEF_QUIK_VNT_ALL_PRS %
%   B31:2/5  DEF_LOAD_ALL  "COMMAND HMI System Load All Defaults" %
%   N21:59  QUICK_VENT_ALL_PRS %
% Rung: 46 %
SOR BST XIC B22:4/8 NXB XIC B31:2/5 BND MOV 5000 N21:60 EOR
%   B22:4/8  DEF_QUIK_VNT_ALL_FLW %
%   B31:2/5  DEF_LOAD_ALL  "COMMAND HMI System Load All Defaults" %
%   N21:60  QUICK_VENT_ALL_FLW %
% Rung: 47 %
SOR BST XIC B22:4/9 NXB XIC B31:2/5 BND MOV 60 N21:61 EOR
%   B22:4/9  DEF_QUIK_BKFL_1_PRS %
%   B31:2/5  DEF_LOAD_ALL  "COMMAND HMI System Load All Defaults" %
%   N21:61  QUICK_BKFIL_1_PRS %
% Rung: 48 %
SOR BST XIC B22:4/10 NXB XIC B31:2/5 BND MOV 5000 N21:62 EOR
%   B22:4/10  DEF_QUIK_BKFL_1_FLW %
%   B31:2/5  DEF_LOAD_ALL  "COMMAND HMI System Load All Defaults" %
%   N21:62  QUICK_BKFIL_1_FLW %
% Rung: 49 %
SOR BST XIC B22:4/11 NXB XIC B31:2/5 BND MOV 20 N21:63 EOR
%   B22:4/11  DEF_QUIK_VNT_A_2_PRS %
%   B31:2/5  DEF_LOAD_ALL  "COMMAND HMI System Load All Defaults" %
%   N21:63  QUICK_VENT_ADS_2_PRS %
% Rung: 50 %
SOR BST XIC B22:4/12 NXB XIC B31:2/5 BND MOV 0 N21:64 EOR
%   B22:4/12  DEF_QUIK_VNT_A_2_FLW %
%   B31:2/5  DEF_LOAD_ALL  "COMMAND HMI System Load All Defaults" %
%   N21:64  QUICK_VENT_ADS_2_FLW %

